// TwinCAT 3 PLC project Untitled1
// ProgramVersion: 3.1.4024.0
// libraries:
//   Tc2_Standard, * (Beckhoff Automation GmbH)
//   Tc2_System, * (Beckhoff Automation GmbH)
//   Tc3_EventLogger, * (Beckhoff Automation GmbH)
//   Tc3_Module, * (Beckhoff Automation GmbH)
// project tree:
//   DUTs/ F_MapSource.TcPOU (not stored)
//   / PlcTask.TcTTO
//   POUs/ FB_SimpleAdsLogEvent_new.TcPOU, MAIN.TcPOU
// real-time tasks:
//   TASK PlcTask: cycle T#10ms, priority 20, ADS port 350

CONFIGURATION Untitled1
    RESOURCE PLC ON TwinCAT3
        TASK PlcTask(INTERVAL := T#10ms, PRIORITY := 20);
        PROGRAM MAIN WITH PlcTask : MAIN;
    END_RESOURCE
END_CONFIGURATION

// ---- POUs/MAIN.TcPOU
PROGRAM MAIN
VAR
	//The FB_SimpleAdsLogEvent_new has the same interface as the FB_SimpleAdsLogEvent sending events via the Tc2 Eventlogger
	//The FB_SimpleAdsLogEvent_new is provided as an sample on how to make use of the resource-representation with the new Eventlogger. 
 	//In combination with the Excel Addin one can migrate the Resource format to the new EventClasses. Please see Infosys for more verbose information 
 
	fbSimpleAdsLogEvent1 : FB_SimpleAdsLogEvent_new;
	bTrigger1: BOOL;
	bQuit1: BOOL;
	
	fbSimpleAdsLogEvent2 : FB_SimpleAdsLogEvent_new;
	bTrigger2: BOOL;
	bQuit2: BOOL;
	
	fbSimpleAdsLogEvent3 : FB_SimpleAdsLogEvent_new;
	bTrigger3: BOOL;
	bQuit3: BOOL;
	
	fbSimpleAdsLogEvent4 : FB_SimpleAdsLogEvent_new;
	bTrigger4: BOOL;
	bQuit4: BOOL;
END_VAR

fbSimpleAdsLogEvent1(
	SourceID:= 1, 
	EventID:= 1, 
	bSetEvent:= bTrigger1, 
	bQuit:= bQuit1, 
	ErrId=> , 
	Error=> );
	
fbSimpleAdsLogEvent2(
	SourceID:= 1, 
	EventID:= 2, 
	bSetEvent:= bTrigger2, 
	bQuit:= bQuit2, 
	ErrId=> , 
	Error=> );
	
fbSimpleAdsLogEvent3(
	SourceID:= 2, 
	EventID:= 1, 
	bSetEvent:= bTrigger3, 
	bQuit:= bQuit3, 
	ErrId=> , 
	Error=> );
	
fbSimpleAdsLogEvent4(
	SourceID:= 2, 
	EventID:= 2, 
	bSetEvent:= bTrigger4, 
	bQuit:= bQuit4, 
	ErrId=> , 
	Error=> );

END_PROGRAM

// ---- POUs/FB_SimpleAdsLogEvent_new.TcPOU
FUNCTION_BLOCK FB_SimpleAdsLogEvent_new
VAR_INPUT
	bSetEvent : BOOL; 
	bQuit : BOOL; 
	SourceID : DINT;  
	EventID : DINT;  
END_VAR
VAR_OUTPUT
	ErrId : UDINT; 
	Error : BOOL;  
END_VAR
VAR
	fb_alarm : FB_TcAlarm; 
	b_InternalSetEvent : BOOL;
    raisingRTrig : R_TRIG;  
	fallingFTrig : F_TRIG;
    clearingRTrig : R_TRIG;  
	e: TcEventEntry;
END_VAR

raisingRTrig(CLK := bSetEvent); 
fallingFTrig(CLK := bSetEvent); 
clearingRTrig(CLK := bQuit); 

// bSetEvent = TRUE -> raise 
IF raisingRTrig.Q AND NOT fb_alarm.bRaised THEN   
  e := F_MapSource(SourceId, EventID);  
  fb_alarm.CreateEx2(e,0); 
  fb_alarm.Raise(0);
END_IF  

// bSetEvent = FALSE -> clear 
IF fallingFTrig.Q AND fb_alarm.bRaised THEN   
  IF(fb_alarm.ipEvent <> 0) THEN 
    ErrId := 0; 
  	fb_alarm.Clear(0);
  ELSE 
	  ErrId := 1; 
  END_IF 
END_IF  

// bQuit = TRUE -> confirm (if ReqMustCon = TRUE) 
IF clearingRTrig.Q AND fb_alarm.bActive THEN   
  IF(fb_alarm.ipEvent <> 0) THEN 
    ErrId := 0; 
  	fb_alarm.Confirm(0);
  ELSE 
	  ErrId := 1; 
  END_IF  
END_IF

END_FUNCTION_BLOCK
